// TwinCAT 3 PLC project IntelligenteWZM_PLCProject
// ProgramVersion: 3.1.4022.4
// libraries:
//   Tc2_Standard, * (Beckhoff Automation GmbH)
//   Tc2_System, * (Beckhoff Automation GmbH)
//   Tc3_Module, * (Beckhoff Automation GmbH)
// project tree:
//   / PlcTask.TcTTO
//   POUs/ GlobaleVariablen.TcGVL, MAIN.TcPOU (not stored)
// real-time tasks:
//   TASK PlcTask: cycle T#10ms, priority 20, ADS port 350
//   TASK Task 1: cycle T#10ms, priority 1, ADS port 301
// I/O:
//   DEVICE Device 2 (EtherCAT), AmsNetId 169.254.30.239.3.1
//     Term 1 (EK1100) [EK1100 EtherCAT Coupler (2A E-Bus)]
//       Term 2 (EL4134) [EL4134 4Ch. Ana. Output -10/+10V, 16bit]
//       Term 3 (EL3104) [EL3104 4Ch. Ana. Input +/-10V Diff.]
//       Term 4 (EL6731-0010) [EL6731-0010 PROFIBUS DP Slave]
//       Term 5 (EL6751) [EL6751 CANopen Master]
//       Term 6 (EL9512) [EL9512 Power supply terminal 12V]
//       Term 11 (EL9011) [EL9011 End Terminal]
//     Term 7 (EK1100) [EK1100 EtherCAT Coupler (2A E-Bus)]
//       Term 8 (EL3632) [EL3632 2Ch. IEPE Sensor]
//       Term 9 (EL3632) [EL3632 2Ch. IEPE Sensor]
//       Term 10 (EL3632) [EL3632 2Ch. IEPE Sensor]
//       Term 12 (EL9011) [EL9011 End Terminal]
//   DEVICE Device 1 (EL6731-0010), AmsNetId 169.254.30.239.2.1
//     Box 1 (EL6731-0010) // Vendor: BECKHOFF Revision: Revision 2.00
//   DEVICE Device 3 (EL6751), AmsNetId 169.254.30.239.4.1
// variable links:
//   IntelligenteWZM_PLCProject/IntelligenteWZM_PLCProject Instance <-> Device 2 (EtherCAT)/Term 7 (EK1100)/Term 8 (EL3632)
//     PlcTask Inputs/GlobaleVariablen.A_OVERSAMPLING_INPUT_1[{0..9}] <-> Ch1 Sample {0..9}/Ch1 Value  (10 links)

CONFIGURATION IntelligenteWZM_PLCProject
    RESOURCE PLC ON TwinCAT3
        TASK PlcTask(INTERVAL := T#10ms, PRIORITY := 20);
        PROGRAM MAIN WITH PlcTask : MAIN;
    END_RESOURCE
END_CONFIGURATION

// ---- POUs/GlobaleVariablen.TcGVL
{attribute 'qualified_only'}
VAR_GLOBAL
	// Eingangssignale aus den Klemmen 
	// Oversampling-Klemmen EL3632
	A_OVERSAMPLING_INPUT_1 AT%I*: ARRAY[0..9] OF INT; // Sensor 1 X 
	A_OVERSAMPLING_INPUT_2 AT%I*: ARRAY[0..9] OF INT; // Sensor 1 Y
	A_OVERSAMPLING_INPUT_3 AT%I*: ARRAY[0..9] OF INT; // Sensor 1 Z
	A_OVERSAMPLING_INPUT_4 AT%I*: ARRAY[0..9] OF INT; // Sensor 2 X
	A_OVERSAMPLING_INPUT_5 AT%I*: ARRAY[0..9] OF INT; // Sensor 2 Y
	A_OVERSAMPLING_INPUT_6 AT%I*: ARRAY[0..9] OF INT; // Sensor 2 Z
END_VAR
